KUKA KRL data list: ConfGarra_NoWait.dat

&ACCESS RVO1
&REL 1
&PARAM EDITMASK = *
DEFDAT ConfGarra_NoWait

ENDDAT
